KUKA KRL program: SET_CP_DAMPING.src

&ACCESS RVO
&REL 6
&PARAM TEMPLATE = C:\KRC\Roboter\Template\FunctionVorgabe
&PARAM EDITMASK = *
DEFFCT BOOL SET_CP_DAMPING( X_VAL:IN, Y_VAL:IN, Z_VAL:IN, A_VAL:IN, B_VAL:IN, C_VAL:IN)

REAL X_VAL, Y_VAL, Z_VAL
REAL A_VAL, B_VAL, C_VAL

$STIFFNESS.CPDAMPING.X = X_VAL
$STIFFNESS.CPDAMPING.Y = Y_VAL
$STIFFNESS.CPDAMPING.Z = Z_VAL
$STIFFNESS.CPDAMPING.A = A_VAL
$STIFFNESS.CPDAMPING.B = B_VAL
$STIFFNESS.CPDAMPING.C = C_VAL

RETURN TRUE

ENDFCT
